{attribute addProperty BoxType "EL2521-0000-1017"}
{attribute addProperty Id "PTO_StatusAT %I*PTO_Status_E3BE96A21620ENC_Status_compactAT %I*ENC_Status_compact_D899538D3240PTO_ControlAT %Q*PTO_Control_0A6210C33240PTO_Target_compactAT %Q*PTO_Target_compact_C80C22BB1620ENC_Control_compactAT %Q*ENC_Control_compact_B20E0FB13240WcStateAT %I*WcState_F855686C1620InfoDataAT %I*InfoData_BC63D37F80100"}
{attribute addProperty CRC "2653298756"}
{attribute addProperty SizeInBites "224"}
{attribute addProperty SizeInBytes "28"}
TYPE EL2521_E52B0EC0 :
STRUCT
	{attribute addProperty Name "PTO_Status"}
	PTO_Status : PTO_Status_E3BE96A2;
	{attribute addProperty Name "ENC_Status_compact"}
	ENC_Status_compact : ENC_Status_compact_D899538D;
	{attribute addProperty Name "PTO_Control"}
	PTO_Control : PTO_Control_0A6210C3;
	{attribute addProperty Name "PTO_Target_compact"}
	PTO_Target_compact : PTO_Target_compact_C80C22BB;
	{attribute addProperty Name "ENC_Control_compact"}
	ENC_Control_compact : ENC_Control_compact_B20E0FB1;
	{attribute addProperty Name "WcState"}
	WcState : WcState_F855686C;
	{attribute addProperty Name "InfoData"}
	InfoData : InfoData_BC63D37F;
END_STRUCT
END_TYPE

(* stored: Version 1.2.0.0, ProductVersion 3.1.4024.9
   DUT EL2521_E52B0EC0: Id {7d51445b-37e7-45c7-a1fe-1cefa0eff3f3} *)
